// TwinCAT 3 PLC project Example_ExecutionToken
// ProgramVersion: 3.1.4024.0
// libraries:
//   Tc3_Module, * (Beckhoff Automation GmbH)
//   ZApplication, 1.6.0.6 (Zeugwerk GmbH)
//   ZAux, 1.6.0.6 (Zeugwerk GmbH)
//   ZCore, 1.6.0.6 (Zeugwerk GmbH)
//   ZEquipment, 1.6.0.6 (Zeugwerk GmbH)
//   ZPlatform, 1.6.0.6 (Zeugwerk GmbH)
// project tree:
//   ZApp/App/ ZApp.TcPOU
//   ZApp/App/_DataTypes/ ZAppStep.TcDUT
//   ZApp/App/_States/ ZAppSequenceBoot.TcPOU, ZAppSequenceBootFault.TcPOU, ZAppSequenceRunning.TcPOU
//   ZApp/App/_SubObjects/ ZAppSequence.TcPOU
//   ZApp/Com/_DataTypes/ ZCom.TcDUT, ZComUnit.TcDUT
//   ZApp/Data/_DataTypes/ ZData.TcDUT, ZDataMachine.TcDUT, ZDataConfig.TcDUT, ZDataCalibration.TcDUT, ZDataRecipe.TcDUT
//   ZApp/Unit/Picker/ IPicker.TcIO, PickerUnit.TcPOU, PickerUnitProgram.TcPOU
//   ZApp/Unit/Picker/_Com/ PickerCom.TcDUT, PickerComPublish.TcDUT, PickerComPublishEquipment.TcDUT, PickerComRef.TcDUT, PickerComRequest.TcDUT, PickerComSubscribe.TcDUT, PickerComSubscribeEquipment.TcDUT
//   ZApp/Unit/Picker/_DataTypes/ PickerState.TcDUT, PickerStep.TcDUT, PickerTokenUsage.TcDUT
//   ZApp/Unit/Picker/_Data/ PickerDataCalibration.TcDUT, PickerDataConfig.TcDUT, PickerDataMachine.TcDUT, PickerDataRef.TcDUT
//   ZApp/Unit/Picker/_Equipment/ PickerActuator.TcPOU, PickerAxis.TcPOU, PickerEquipment.TcPOU, PickerFieldbus.TcPOU, PickerIo.TcPOU, PickerLinkedUnit.TcPOU
//   ZApp/Unit/Picker/_States/ PickerSequenceAutomatic.TcPOU, PickerSequenceBoot.TcPOU, PickerSequenceFaultReaction.TcPOU, PickerSequenceGoHome.TcPOU, PickerSequenceStop.TcPOU
//   ZApp/Unit/Picker/_SubObjects/ PickerContainer.TcPOU, PickerSequence.TcPOU
//   ZApp/ ZGlobal.TcGVL, ZModuleProgram.TcPOU, ZModuleTask.TcTTO
// real-time tasks:
//   TASK ZModuleTask: cycle T#10ms, priority 20, ADS port 350

CONFIGURATION Example_ExecutionToken
    RESOURCE PLC ON TwinCAT3
        TASK ZModuleTask(INTERVAL := T#10ms, PRIORITY := 20);
        PROGRAM ZModuleProgram WITH ZModuleTask : ZModuleProgram;
    END_RESOURCE
END_CONFIGURATION

// ---- ZApp/App/_DataTypes/ZAppStep.TcDUT
{attribute 'qualified_only'}
{attribute 'to_string'}
TYPE ZAppStep :
(
  Undefined := 0
  
  ,BootBegin
  ,BootLoadDefaultData
  ,BootEnd
  ,BootFaultBegin
  ,BootFaultEnd 
  ,RunningBegin
  ,RunningEnd   
);
END_TYPE

// ---- ZApp/Com/_DataTypes/ZCom.TcDUT
TYPE ZCom :
STRUCT
  // module context
  App : ZApplication.ApplicationComPublish;
  Alarming : ZApplication.AlarmingCom;
  Messages : ZApplication.MessagingCom;
  
  // unit context
  Unit : ZComUnit;

END_STRUCT
END_TYPE

// ---- ZApp/Com/_DataTypes/ZComUnit.TcDUT
TYPE ZComUnit :
STRUCT
{region "Picker"}
{IF NOT (defined (Picker_disabled))}
  Picker : PickerCom;
  {attribute 'ZId' := 'c43c28b7-9e8c-48c6-a4f8-946be27888d3'}
{END_IF}
{endregion}
{attribute '__ZwPlcApplicationComUnitDeclaration__'} // Do not remove this attribute! It is used for code generation.
END_STRUCT
END_TYPE

// ---- ZApp/Data/_DataTypes/ZData.TcDUT
TYPE ZData :
STRUCT
  Config : ZDataConfig;
  Machine : ZDataMachine;
  Calibration : ZDataCalibration;
  Recipe : ZDataRecipe;
END_STRUCT
END_TYPE

// ---- ZApp/Data/_DataTypes/ZDataMachine.TcDUT
TYPE ZDataMachine :
STRUCT
{region "Picker"}
{IF NOT (defined (Picker_disabled))}
  Picker : PickerDataMachine;
  {attribute 'ZId' := 'c43c28b7-9e8c-48c6-a4f8-946be27888d3'}
{END_IF}
{endregion}
{attribute '__ZwPlcApplicationDataMachineDeclaration__'} // Do not remove this attribute! It is used for code generation.
END_STRUCT
END_TYPE

// ---- ZApp/Data/_DataTypes/ZDataConfig.TcDUT
TYPE ZDataConfig :
STRUCT
{region "Picker"}
{IF NOT (defined (Picker_disabled))}
  Picker : PickerDataConfig;
  {attribute 'ZId' := 'c43c28b7-9e8c-48c6-a4f8-946be27888d3'}
{END_IF}
{endregion}
{attribute '__ZwPlcApplicationDataConfigDeclaration__'} // Do not remove this attribute! It is used for code generation.
END_STRUCT
END_TYPE

// ---- ZApp/Data/_DataTypes/ZDataCalibration.TcDUT
TYPE ZDataCalibration :
STRUCT
{region "Picker"}
{IF NOT (defined (Picker_disabled))}
  Picker : PickerDataCalibration;
  {attribute 'ZId' := 'c43c28b7-9e8c-48c6-a4f8-946be27888d3'}
{END_IF}
{endregion}
{attribute '__ZwPlcApplicationDataCalibrationDeclaration__'} // Do not remove this attribute! It is used for code generation.
END_STRUCT
END_TYPE

// ---- ZApp/Data/_DataTypes/ZDataRecipe.TcDUT
TYPE ZDataRecipe :
STRUCT
  RecipeParam1 : LREAL;
  RecipeParam2 : LREAL;
  RecipeParam3 : LREAL;
END_STRUCT
END_TYPE

// ---- ZApp/Unit/Picker/_Com/PickerCom.TcDUT
/// This struct contains variables that
/// * are read from outside (e.g. HMI) to retrieve information about the unit's current state and (temporary) parameters (= `publish`) 
/// * are written from outside (e.g. HMI) to control the unit via ADS (= `subscribe`) 
TYPE PickerCom :
STRUCT
  Publish : PickerComPublish;
  Subscribe : PickerComSubscribe;
END_STRUCT
END_TYPE

// ---- ZApp/Unit/Picker/_Com/PickerComPublish.TcDUT
/// this is the container of informations that the unit wants to share with the world outside of the PLC
/// This struct should only be read from by external applications.
TYPE PickerComPublish :
STRUCT
  State : ZApplication.UnitStateMachineState; // state the unit is in
  Request : PickerComRequest; // booleans that indictate which action is currently possible to perform with this unit
  Equipment : PickerComPublishEquipment;  // structs for equipment objects which are used by the bridges
END_STRUCT
END_TYPE

// ---- ZApp/Unit/Picker/_Com/PickerComPublishEquipment.TcDUT
TYPE PickerComPublishEquipment :
STRUCT

{region "Vertical : Axis"}
  Vertical : ZApplication.AxisComPublish;
  {attribute 'ZId' := '1181714e-d83e-4cf6-aa91-287de19a3556'}
{endregion}

{attribute '__ZwPlcUnitComDeclaration__'} // Do not remove this attribute! It is used for code generation.

END_STRUCT
END_TYPE

// ---- ZApp/Unit/Picker/_Com/PickerComRef.TcDUT
/// container for all communication data types that are used by the unit
TYPE PickerComRef :
STRUCT
  Publish : REFERENCE TO PickerComPublish; 
  Subscribe : REFERENCE TO PickerComSubscribe; 
END_STRUCT
END_TYPE

// ---- ZApp/Unit/Picker/_Com/PickerComRequest.TcDUT
TYPE PickerComRequest :
STRUCT
  Start : BOOL;
  Stop : BOOL;
  GoHome : BOOL;
  Halt : BOOL;
END_STRUCT
END_TYPE

// ---- ZApp/Unit/Picker/_Com/PickerComSubscribe.TcDUT
TYPE PickerComSubscribe :
STRUCT
  Request : PickerComRequest; // contains booleans that are used to start a specific sequence.
  Equipment : PickerComSubscribeEquipment;  // structs for equipment objects which are used by the bridges
END_STRUCT
END_TYPE

// ---- ZApp/Unit/Picker/_Com/PickerComSubscribeEquipment.TcDUT
TYPE PickerComSubscribeEquipment :
STRUCT

{region "Vertical : Axis"}
  Vertical : ZApplication.AxisComSubscribe;
  {attribute 'ZId' := '1181714e-d83e-4cf6-aa91-287de19a3556'}
{endregion}

{attribute '__ZwPlcUnitComDeclaration__'} // Do not remove this attribute! It is used for code generation.

END_STRUCT
END_TYPE

// ---- ZApp/Unit/Picker/_DataTypes/PickerState.TcDUT
/// This enumeration contains all used defined sequences of a unit.
/// Per default a unit makes use of the states that are contained in (UnitStateDefault)[xref:ZApplication.UnitStateDefault]. However,
/// most of the time a unit need to perform some application depend sequences that can be performed by putting the unit into userdefined states.
/// For instance, a robotic unit could use the state (automatic)[xref:ZApplication.UnitStateDefault] to lift an object from point A to point B,
/// a userdefined state could be used to open and close the robotic-units gripper, respectively
{attribute 'qualified_only'}
TYPE PickerState :
(
	UserdefinedState1 := ZApplication.UnitStateMachineState.Last+1
);
END_TYPE

// ---- ZApp/Unit/Picker/_DataTypes/PickerStep.TcDUT
/// This enumeration contains all steps that are used by the various sequences of a unit.
/// Sequences use a subrange (***Begin to ***End) of this enumeration.
{attribute 'qualified_only'}
{attribute 'to_string'}
TYPE PickerStep :
(
  Undefined := 0
  
  ,BootBegin
  ,BootEnd 

  ,StopBegin
  ,StopEnd

  ,AutomaticBegin
  ,AutomaticEnd
  
  ,GoHomeBegin
  ,GoHomeMoveAxisTo60
  ,GoHomeMoveAxisBackTo0
  ,GoHomeEnd 
  
  ,FaultReactionBegin
  ,FaultReactionEnd
);
END_TYPE

// ---- ZApp/Unit/Picker/_DataTypes/PickerTokenUsage.TcDUT
{attribute 'qualified_only'}
TYPE PickerTokenUsage :
(
	StartToken
  ,ExecutionToken
  ,SequenceAsToken
);
END_TYPE

// ---- ZApp/Unit/Picker/_Data/PickerDataCalibration.TcDUT
/// calibration that is determined by calibration sequences of the unit (static offsets, shifts)
TYPE PickerDataCalibration :
STRUCT
END_STRUCT
END_TYPE

// ---- ZApp/Unit/Picker/_Data/PickerDataConfig.TcDUT
/// configuration data that is used during boot to configure the Units equipment
TYPE PickerDataConfig :
STRUCT
  Simulated : BOOL;
END_STRUCT
END_TYPE

// ---- ZApp/Unit/Picker/_Data/PickerDataMachine.TcDUT
/// machine data that is used through most sequences of the unit (motor speed, axes positions, ...)
TYPE PickerDataMachine :
STRUCT
  Slowspeed : LREAL;
  Highspeed : LREAL;
END_STRUCT
END_TYPE

// ---- ZApp/Unit/Picker/_Data/PickerDataRef.TcDUT
/// container for all data that are used by the unit
TYPE PickerDataRef :
STRUCT
  Config : REFERENCE TO PickerDataConfig; // data required for booting the unit (axes configuration, simulation, parameters that have to be written in PREOP, ...)
  Machine : REFERENCE TO PickerDataMachine; // speeds, positions, ...
  Calibration : REFERENCE TO PickerDataCalibration; // offsets, shifts of nominal to actual values
END_STRUCT
END_TYPE

// ---- ZApp/ZGlobal.TcGVL
{attribute 'qualified_only'}
VAR_GLOBAL
  Com : ZCom;
END_VAR
VAR_GLOBAL PERSISTENT
  Data : ZData;
END_VAR

// ---- ZApp/Unit/Picker/IPicker.TcIO
INTERFACE IPicker EXTENDS ZApplication.IUnit

END_INTERFACE

// ---- ZApp/ZModuleProgram.TcPOU
/// Zeugwerk Application
PROGRAM ZModuleProgram
VAR_INPUT
{region "ZModuleProgram : Utility"}
  App : ZApp(displayName:='Zeugwerk-Application Template', com:=ZGlobal.Com.App);
  Datetime : ZAux.DateTimeUM;
  {attribute 'ZId' := ''}
{endregion}
{region "ZModuleProgram : Logging"}
  Alarming : ZApplication.Alarming(App, datetime := Datetime, com := ZGlobal.Com.Alarming);
  LoggerHmi : ZApplication.Messaging(App, datetime := Datetime, com := ZGlobal.Com.Messages);
  LoggerFile : ZAux.LoggerFile7FF(App, datetime := Datetime, filePath:='C:\Zeugwerk\logs\messages.log', target:='');
  Logger : ZAux.Logging;
  {attribute 'ZId' := ''}
{endregion}  
{attribute '__ZwPlcApplicationModuleProgramDeclaration__'} // Do not remove this attribute! It is used for code generation.
{region "Picker"}
{undefine RunInSeparateProgram}
{IF NOT (defined (Picker_disabled)) AND NOT (defined (RunInSeparateProgram))}
  Picker : PickerUnit(displayName := 'Picker', // name of the unit (for logging)
					  parent := App, // caller of the Unit's cyclic method. If the Unit runs in its own context use 0
						configdata := ZGlobal.Data.Config.Picker,
						machinedata := ZGlobal.Data.Machine.Picker,
						calibrationdata := ZGlobal.Data.Calibration.Picker,
						com := ZGlobal.Com.Unit.Picker);
  {attribute 'section' := '__ZwPlcUnitProgramDeclaration__'}
  {attribute 'ZId' := 'c43c28b7-9e8c-48c6-a4f8-946be27888d3'}
{END_IF}
{endregion}
{attribute '__ZwPlcUnitProgramDeclaration__'} // Do not remove this attribute! It is used for code generation.
END_VAR

{region "ZModuleProgram : Utility"}
  Datetime.Cyclic();
  App.Cyclic();
  {attribute 'ZId' := ''}
{endregion}
{attribute '__ZwPlcApplicationModuleProgramImplementation__'} // Do not remove this attribute! It is used for code generation.

END_PROGRAM

// ---- ZApp/App/ZApp.TcPOU
FUNCTION_BLOCK ZApp EXTENDS ZApplication.Application
VAR
  _boot : ZAppSequenceBoot;
  _bootFault : ZAppSequenceBootFault;
  _running : ZAppSequenceRunning;
END_VAR

METHOD FB_init : BOOL
VAR_INPUT
  bInitRetains : BOOL; /// if TRUE, the retain variables are initialized (warm start / cold start)
  bInCopyCode : BOOL; /// if TRUE, the instance afterwards gets moved into the copy code (online change)
  displayName : ZCore.ZString;
  com : REFERENCE TO ZApplication.ApplicationComPublish;
END_VAR
SetBootSequence(_boot);
SetBootFaultSequence(_bootFault);
SetRunningSequence(_running);
END_METHOD

END_FUNCTION_BLOCK

// ---- ZApp/App/_States/ZAppSequenceBoot.TcPOU
FUNCTION_BLOCK ZAppSequenceBoot EXTENDS ZAppSequence IMPLEMENTS ZCore.ISequence
VAR
  _step : ZCore.Step(ZAppStep.BootBegin, ZAppStep.BootEnd);
END_VAR

IF OnStart(_step)
THEN
  // init custom sequence variables here ...
END_IF

REPEAT
  LogStep();

  CASE _step.Index OF
    (* -------------------------------------------------------------------------------------------------------------------------------- *)
    ZAppStep.BootBegin:
    (* -------------------------------------------------------------------------------------------------------------------------------- *)
    
      IF _step.OnEntry()
      THEN
        ZModuleProgram.LoggerFile.MinimumLevel := ZCore.LogLevel.Trace;
        ZModuleProgram.Logger.AddLogger(ZModuleProgram.LoggerFile);        
        {attribute '__ZwPlcAppZComModuleContext__'} // Do not remove this attribute! It is used for code generation.      
      END_IF
      
	  IF ZModuleProgram.Datetime.State <> ZCore.ObjectState.Booting
      THEN
        _step.SetNext(ZAppStep.BootLoadDefaultData);        
      END_IF
      
    (* -------------------------------------------------------------------------------------------------------------------------------- *)
    ZAppStep.BootLoadDefaultData:
    (* -------------------------------------------------------------------------------------------------------------------------------- *)

      {warning 'The application is loading the default config data on every restart!'}
      LoadDefaultConfigData();
      
      IF IsCommissioning()
      THEN
        LoadDefaultData();
      END_IF
      
      _step.SetNext(ZAppStep.BootEnd);
      
    (* -------------------------------------------------------------------------------------------------------------------------------- *)
    ZAppStep.BootEnd:
    (* -------------------------------------------------------------------------------------------------------------------------------- *)
      SetBusy(FALSE);
      
  ELSE
    Abort('sequence contains unhandled step');
  END_CASE
UNTIL _step.IsNotRepeatable() OR_ELSE NOT Busy END_REPEAT

METHOD  IsCommissioning : BOOL
IsCommissioning := TRUE;
END_METHOD

METHOD FINAL LoadDefaultConfigData

{region "Picker"}
  {IF NOT (defined (Picker_disabled))}
  ZGlobal.Data.Config.Picker.Simulated := TRUE;
  {region "UserInitCode"}
  // put your individual init code for this unit here
  {endregion}
  {END_IF}
  {attribute 'ZId' := 'c43c28b7-9e8c-48c6-a4f8-946be27888d3'}
{endregion}

{attribute '__ZwPlcUnitLoadDefaultConfigData__'} // Do not remove this attribute! It is used for code generation.
END_METHOD

METHOD FINAL LoadDefaultData

{attribute '__ZwPlcUnitLoadDefaultData__'} // Do not remove this attribute! It is used for code generation.
END_METHOD

END_FUNCTION_BLOCK

// ---- ZApp/App/_SubObjects/ZAppSequence.TcPOU
FUNCTION_BLOCK ABSTRACT ZAppSequence EXTENDS ZApplication.Sequence IMPLEMENTS ZCore.ISequence

METHOD StepDecoded : ZCore.ZString
VAR_INPUT
  stepIndex : INT;
END_VAR
VAR_INST
  _stepIndexDecoded : ZAppStep;
END_VAR
_stepIndexDecoded := stepIndex;
StepDecoded := TO_STRING(_stepIndexDecoded);
END_METHOD

END_FUNCTION_BLOCK

// ---- ZApp/App/_States/ZAppSequenceBootFault.TcPOU
FUNCTION_BLOCK ZAppSequenceBootFault EXTENDS ZAppSequence IMPLEMENTS ZCore.ISequence
VAR
  _step : ZCore.Step(ZAppStep.BootFaultBegin, ZAppStep.BootFaultEnd);
END_VAR

IF OnStart(_step)
THEN
  // init custom sequence variables here ...
END_IF

REPEAT
  LogStep();

  CASE _step.Index OF
    (* -------------------------------------------------------------------------------------------------------------------------------- *)
    ZAppStep.BootFaultBegin:
    (* -------------------------------------------------------------------------------------------------------------------------------- *)
      _step.SetNext(ZAppStep.BootFaultEnd);
      
    (* -------------------------------------------------------------------------------------------------------------------------------- *)
    ZAppStep.BootFaultEnd:
    (* -------------------------------------------------------------------------------------------------------------------------------- *)
      SetBusy(FALSE);
      
  ELSE
    Abort('sequence contains unhandled step');
  END_CASE
UNTIL _step.IsNotRepeatable() OR_ELSE NOT Busy END_REPEAT

END_FUNCTION_BLOCK

// ---- ZApp/App/_States/ZAppSequenceRunning.TcPOU
FUNCTION_BLOCK ZAppSequenceRunning EXTENDS ZAppSequence IMPLEMENTS ZCore.ISequence
VAR
  _step : ZCore.Step(ZAppStep.RunningBegin, ZAppStep.RunningEnd);
END_VAR

IF OnStart(_step)
THEN
  // init custom sequence variables here ...
END_IF

REPEAT
  LogStep();

  CASE _step.Index OF
    (* -------------------------------------------------------------------------------------------------------------------------------- *)
    ZAppStep.RunningBegin:
    (* -------------------------------------------------------------------------------------------------------------------------------- *)
      ; // implement me
      
    (* -------------------------------------------------------------------------------------------------------------------------------- *)
    ZAppStep.RunningEnd:
    (* -------------------------------------------------------------------------------------------------------------------------------- *)
      SetBusy(FALSE);
      
  ELSE
    Abort('sequence contains unhandled step');
  END_CASE
UNTIL _step.IsNotRepeatable() OR_ELSE NOT Busy END_REPEAT

END_FUNCTION_BLOCK

// ---- ZApp/Unit/Picker/PickerUnit.TcPOU
/// Declaration of a distinct unit of this application
FUNCTION_BLOCK PickerUnit EXTENDS ZApplication.Unit IMPLEMENTS IPicker
VAR
  _equipment : PickerEquipment(THIS^);
  _data : PickerDataRef;
  _com : PickerComRef;

  _boot : PickerSequenceBoot(THIS^);
  _automatic : PickerSequenceAutomatic(THIS^);
  _stop : PickerSequenceStop(THIS^);
  _gohome : PickerSequenceGoHome(THIS^);
  _faultReaction : PickerSequenceFaultReaction(THIS^);
  
  _statemachine : ZApplication.UnitStateMachine;

  _observeTimer : ZAux.Timer;
END_VAR

{attribute 'ZId' := '91d6f29c-305c-4899-88ef-1e5d578c2af4'}

IF _observeTimer.Done THEN
  _observeTimer.WaitAsync(0.1);
  
  // monitor _com for requested actions (e.g. start homing, start automatic mode, ...)
  ObserveRequest(_com.Subscribe.Request.Start, ZApplication.UnitStateMachineState.Automatic);
  ObserveRequest(_com.Subscribe.Request.Stop, ZApplication.UnitStateMachineState.Stop);
  ObserveRequest(_com.Subscribe.Request.GoHome, ZApplication.UnitStateMachineState.GoHome);
  ObserveRequest(_com.Subscribe.Request.Halt, ZApplication.UnitStateMachineState.Halt);
  
  // provide relevant information via ADS
  _com.Publish.Request.Stop := _stateMachine.IsTransitionAllowed(ZApplication.UnitStateMachineState.Stop);
  _com.Publish.Request.Start := _stateMachine.IsTransitionAllowed(ZApplication.UnitStateMachineState.Automatic);
  _com.Publish.Request.GoHome := _stateMachine.IsTransitionAllowed(ZApplication.UnitStateMachineState.GoHome);
  _com.Publish.Request.Halt := _stateMachine.IsTransitionAllowed(ZApplication.UnitStateMachineState.Halt);

  _com.Publish.State := _stateMachine.State();
END_IF

METHOD FB_init : BOOL
VAR_INPUT
  bInitRetains : BOOL; // if TRUE, the retain variables are initialized (warm start / cold start)
  bInCopyCode : BOOL;  // if TRUE, the instance afterwards gets moved into the copy code (online change)
  parent : ZCore.IManagedObject; // caller of the Unit's cyclic method. If the Unit runs in its own context use 0
  displayName : ZCore.ZString;  // name of this unit as it should show up in the logger
  configdata : REFERENCE TO PickerDataConfig;  // reference to the configuration data that is used during boot to configure the Units equipment
  machinedata : REFERENCE TO PickerDataMachine; // reference to the machine data that is used through most sequences of the unit (motor speed, axes positions, ...)
  calibrationdata : REFERENCE TO PickerDataCalibration;  // reference to calibration that is determined by calibration sequences of the unit (static offsets, shifts)
  com : REFERENCE TO PickerCom;  // reference to the communication interface that is used to control this Unit via ADS
END_VAR
_name := displayName;

// initialize local logger decorator
_loggerDecorator.FB_init(bInitRetains, bInCopyCode, _name, ZModuleProgram.Logger);
_alarmingDecorator.FB_init(bInitRetains, bInCopyCode, _name, ZModuleProgram.Alarming);

// setup data
_data.Config REF= configdata;
_data.Machine REF= machinedata;
_data.Calibration REF= calibrationdata;
_com.Publish REF= com.Publish;
_com.Subscribe REF= com.Subscribe;

// ------- sequence initialization, map sequences of this unit to the statemachine -------
{attribute '__ZwPlcUnitInitSequenceImplementation__'} // Do not remove this attribute! It is used for code generation.
_statemachine.SetSequence(ZApplication.UnitStateMachineState.Boot, _boot);
_statemachine.SetSequence(ZApplication.UnitStateMachineState.FaultReaction, _faultReaction);
_statemachine.SetSequence(ZApplication.UnitStateMachineState.Gohome, _gohome);
_statemachine.SetSequence(ZApplication.UnitStateMachineState.Stop, _stop);
_statemachine.SetSequence(ZApplication.UnitStateMachineState.Automatic, _automatic);

_statemachine.SetName(_name);
_statemachine.SetLogger(_logger);

// set initial state
_statemachine.SetState(ZApplication.UnitStateMachineState.Boot);
SetStateMachine(_statemachine);
END_METHOD

END_FUNCTION_BLOCK

// ---- ZApp/Unit/Picker/_Equipment/PickerEquipment.TcPOU
/// This function block is a container for equipment that is used by this unit.
/// Equipment is grouped by its kind (actuator, axes, io, ...).
/// It extends from [ManagedObjectContainer](xref:ZCore.ManagedObjectContainer) such that the parent
/// (= the unit itself) can be passed to equipment instances.
FUNCTION_BLOCK PickerEquipment EXTENDS PickerContainer
VAR_INPUT
  Io : PickerIo(_parent);
  Actuator : PickerActuator(_parent);
  Axis : PickerAxis(_parent);
  Fieldbus : PickerFieldbus(_parent);
  Unit : PickerLinkedUnit(_parent);
END_VAR

END_FUNCTION_BLOCK

// ---- ZApp/Unit/Picker/_SubObjects/PickerContainer.TcPOU
FUNCTION_BLOCK PickerContainer EXTENDS ZCore.ObjectContainer
VAR_INPUT
END_VAR
VAR_OUTPUT
END_VAR
VAR
  {attribute 'hide'}
  _parent : REFERENCE TO PickerUnit;
END_VAR

{attribute 'hide' }
METHOD FB_init : BOOL
VAR_INPUT
	bInitRetains : BOOL; // if TRUE, the retain variables are initialized (warm start / cold start)
	bInCopyCode : BOOL;  // if TRUE, the instance afterwards gets moved into the copy code (online change)
  unit : REFERENCE TO PickerUnit;
END_VAR
_parent REF= unit;
END_METHOD

END_FUNCTION_BLOCK

// ---- ZApp/Unit/Picker/_Equipment/PickerIo.TcPOU
/// This function block is a container for all I/Os that are used by this unit.
/// The parent of all objects can be directly transfered in their constructor (this is only relevant for equipment objects
/// that have to be managed (e.g. [DebouncedInput](xref:ZEquipment.DebouncedInput), [Light](xref:ZEquipment.Light), ...).
FUNCTION_BLOCK PickerIo EXTENDS PickerContainer
VAR
  {attribute 'hide'}
  _iobridge : ZApplication.IoBridge(_parent);
END_VAR
VAR_INPUT

{attribute '__ZwPlcUnitEquipmentDeclaration__'} // Do not remove this attribute! It is used for code generation.
END_VAR

IF _isInitialized
THEN
  RETURN;
END_IF

  _iobridge.SetLogger(_parent._logger);

{attribute '__ZwPlcUnitEquipmentImplementation__'} // Do not remove this attribute! It is used for code generation.

_isInitialized := TRUE;

END_FUNCTION_BLOCK

// ---- ZApp/Unit/Picker/_Equipment/PickerActuator.TcPOU
/// This function block is a container for all actuator objects that are used by this unit.
/// The parent of all objects can be directly transfered in their constructor (this is only relevant for equipment objects
/// that have to be managed (e.g. [DebouncedInput](xref:ZEquipment.DebouncedInput), [Light](xref:ZEquipment.Light), ...).
FUNCTION_BLOCK PickerActuator EXTENDS PickerContainer
VAR
  {attribute 'hide'}
  _actuatorbridge : ZApplication.ActuatorBridge(_parent);
  {attribute 'hide'}
  _iobridge : ZApplication.IoBridge(_parent);
END_VAR
VAR_INPUT

{attribute '__ZwPlcUnitEquipmentDeclaration__'} // Do not remove this attribute! It is used for code generation.
END_VAR

IF _isInitialized
THEN
  RETURN;
END_IF

  _actuatorbridge.SetLogger(_parent._logger);

{attribute '__ZwPlcUnitEquipmentImplementation__'} // Do not remove this attribute! It is used for code generation.

_isInitialized := TRUE;

END_FUNCTION_BLOCK

// ---- ZApp/Unit/Picker/_Equipment/PickerAxis.TcPOU
/// This function block is a container for all axis objects that are used by this unit.
/// The parent of all objects can be directly transfered in their constructor (this is only relevant for equipment objects
/// that have to be managed (e.g. [DebouncedInput](xref:ZEquipment.DebouncedInput), [Light](xref:ZEquipment.Light), ...).
FUNCTION_BLOCK PickerAxis EXTENDS PickerContainer
VAR
  {attribute 'hide'}
  _axisbridge : ZApplication.AxisBridge(_parent);
END_VAR
VAR_INPUT

{region "Vertical : AxisPlcOpenMc"}
  Vertical : ZEquipment.AxisPlcOpenMc(_parent);
  {attribute 'ZId' := '1181714e-d83e-4cf6-aa91-287de19a3556'}
{endregion}

{attribute '__ZwPlcUnitEquipmentDeclaration__'} // Do not remove this attribute! It is used for code generation.
END_VAR

IF _isInitialized
THEN
  RETURN;
END_IF

  _axisbridge.SetLogger(_parent._logger);

{region "Vertical : AxisPlcOpenMc"}
  Vertical.SetLogger(_parent._logger);
  Vertical.SetName(name:='Vertical');
  Vertical.SetSimulation(_parent._data.Config.Simulated);
  _axisbridge.AddAxisPlcOpenMc(axis:=Vertical, publish:=_parent._com.Publish.Equipment.Vertical, subscribe:=_parent._com.Subscribe.Equipment.Vertical);

  {region "UserInitCode"}
  // put your individual init code for this Axis here
  {endregion}

  {attribute 'ZId' := '1181714e-d83e-4cf6-aa91-287de19a3556'}
{endregion}

{attribute '__ZwPlcUnitEquipmentImplementation__'} // Do not remove this attribute! It is used for code generation.

_isInitialized := TRUE;

END_FUNCTION_BLOCK

// ---- ZApp/Unit/Picker/_Equipment/PickerFieldbus.TcPOU
/// This function block is a container for all axis objects that are used by this unit.
/// The parent of all objects can be directly transfered in their constructor (this is only relevant for equipment objects
/// that have to be managed (e.g. [DebouncedInput](xref:ZEquipment.DebouncedInput), [Light](xref:ZEquipment.Light), ...).
FUNCTION_BLOCK PickerFieldbus EXTENDS PickerContainer
VAR
END_VAR
VAR_INPUT

{attribute '__ZwPlcUnitEquipmentDeclaration__'} // Do not remove this attribute! It is used for code generation.
END_VAR

IF _isInitialized
THEN
  RETURN;
END_IF

{attribute '__ZwPlcUnitEquipmentImplementation__'} // Do not remove this attribute! It is used for code generation.

_isInitialized := TRUE;

END_FUNCTION_BLOCK

// ---- ZApp/Unit/Picker/_Equipment/PickerLinkedUnit.TcPOU
/// This function block is a container for all linked units that are used by this unit.
/// Linked units can be addressed through their individual interface.
FUNCTION_BLOCK PickerLinkedUnit EXTENDS PickerContainer
VAR_INPUT

{attribute '__ZwPlcUnitEquipmentDeclaration__'} // Do not remove this attribute! It is used for code generation.
END_VAR

IF _isInitialized
THEN
  RETURN;
END_IF

{attribute '__ZwPlcUnitEquipmentImplementation__'} // Do not remove this attribute! It is used for code generation.

_isInitialized := TRUE;

END_FUNCTION_BLOCK

// ---- ZApp/Unit/Picker/_States/PickerSequenceBoot.TcPOU
FUNCTION_BLOCK PickerSequenceBoot EXTENDS PickerSequence IMPLEMENTS ZCore.ISequence
VAR
  _step : ZCore.Step(PickerStep.BootBegin, PickerStep.BootEnd);
END_VAR

IF OnStart(_step) THEN
  ; // init custom sequence variables here ...
END_IF

REPEAT
  LogStep();

  CASE _step.Index OF
    (* -------------------------------------------------------------------------------------------------------------------------------- *)
    PickerStep.BootBegin:
    (* -------------------------------------------------------------------------------------------------------------------------------- *)
      IF _step.OnEntry()
      THEN
        // initialize equipment
        _io();
        _actuator();
        _fieldbus();
        _axis();
        _unit();
      END_IF
      
      _parent._objectManager.Cyclic();      
      Assert(_parent._objectManager);
      IF _parent._objectManager.Booted
      THEN
        _step.SetNext(PickerStep.BootEnd);
      END_IF

    (* -------------------------------------------------------------------------------------------------------------------------------- *)
    PickerStep.BootEnd:
    (* -------------------------------------------------------------------------------------------------------------------------------- *)
      SetBusy(FALSE);
      
  ELSE
    Abort('sequence contains unhandled step');
  END_CASE
UNTIL _step.IsNotRepeatable() OR_ELSE NOT Busy END_REPEAT

END_FUNCTION_BLOCK

// ---- ZApp/Unit/Picker/_SubObjects/PickerSequence.TcPOU
FUNCTION_BLOCK PickerSequence EXTENDS ZApplication.Sequence
VAR
  {attribute 'hide'}
  _parent : REFERENCE TO PickerUnit;
  _io : REFERENCE TO PickerIo;
  _actuator : REFERENCE TO PickerActuator;
  _fieldbus : REFERENCE TO PickerFieldbus;
  _axis : REFERENCE TO PickerAxis;
  _data : REFERENCE TO PickerDataRef;
  _unit : REFERENCE TO PickerLinkedUnit;  
END_VAR

METHOD FB_init : BOOL
VAR_INPUT
  bInitRetains : BOOL; // if TRUE, the retain variables are initialized (warm start / cold start)
  bInCopyCode : BOOL;  // if TRUE, the instance afterwards gets moved into the copy code (online change)
  unit : REFERENCE TO PickerUnit;
END_VAR
_parent REF= unit;
_alarming := unit._alarming;
_io REF= unit._equipment.Io;
_actuator REF= unit._equipment.Actuator;
_fieldbus REF= unit._equipment.Fieldbus;
_axis REF= unit._equipment.Axis;
_unit REF= unit._equipment.Unit;
_data REF= unit._data;
_loggerDiagnostics.SetLogger(unit._logger);
END_METHOD

METHOD StepDecoded : ZCore.ZString
VAR_INPUT
  stepIndex : INT;
END_VAR
VAR_INST
  _stepIndexDecoded : PickerStep;
END_VAR
_stepIndexDecoded := stepIndex;
stepDecoded := TO_STRING(_stepIndexDecoded);
END_METHOD

END_FUNCTION_BLOCK

// ---- ZApp/Unit/Picker/_States/PickerSequenceAutomatic.TcPOU
FUNCTION_BLOCK PickerSequenceAutomatic EXTENDS PickerSequence IMPLEMENTS ZCore.ISequence
VAR
  _step : ZCore.Step(PickerStep.AutomaticBegin, PickerStep.AutomaticEnd);
END_VAR

IF NOT Busy THEN
  RETURN;
END_IF

IF OnStart(_step) THEN
  ; // init custom sequence variables here ...
END_IF

IF OnStop() THEN
  RETURN; // external stop was triggered
END_IF

IF OnHalt() THEN
  ; // Halting := TRUE; // Uncomment to acknowledge that the sequence is halting
END_IF

REPEAT
  LogStep();

  CASE _step.Index OF
    (* -------------------------------------------------------------------------------------------------------------------------------- *)
    PickerStep.AutomaticBegin:
    (* -------------------------------------------------------------------------------------------------------------------------------- *)
      IF _step.OnEntry()
      THEN
        ;
      END_IF

      // Await(obj1:=, nextStep:=PickerStep.AutomaticEnd);
      _step.SetNext(PickerStep.AutomaticEnd);
    
    (* -------------------------------------------------------------------------------------------------------------------------------- *)
    PickerStep.AutomaticEnd:
    (* -------------------------------------------------------------------------------------------------------------------------------- *)
      SetBusy(FALSE);
  
  ELSE
    Abort('sequence contains unhandled step');
  END_CASE
UNTIL _step.IsNotRepeatable() OR_ELSE NOT Busy END_REPEAT

END_FUNCTION_BLOCK

// ---- ZApp/Unit/Picker/_States/PickerSequenceStop.TcPOU
FUNCTION_BLOCK PickerSequenceStop EXTENDS PickerSequence IMPLEMENTS ZCore.ISequence
VAR
  _step : ZCore.Step(PickerStep.StopBegin, PickerStep.StopEnd);
  _timerSim : ZAux.Timer;
END_VAR

IF OnStart(_step) THEN
  ; // init custom sequence variables here ...
END_IF

REPEAT
  LogStep();

  CASE _step.Index OF
    (* -------------------------------------------------------------------------------------------------------------------------------- *)
    PickerStep.StopBegin:
    (* -------------------------------------------------------------------------------------------------------------------------------- *)
      IF _step.OnEntry()
      THEN
        _timerSim.WaitAsync(5);
			END_IF
      
      Await(_timerSim, nextStep:=PickerStep.StopEnd);
      // _step.SetNext(index:=PickerStep.StopEnd);

    (* -------------------------------------------------------------------------------------------------------------------------------- *)
    PickerStep.StopEnd:
    (* -------------------------------------------------------------------------------------------------------------------------------- *)    
      SetBusy(FALSE);
  
  ELSE
    Abort('sequence contains unhandled step');
  END_CASE
UNTIL _step.IsNotRepeatable() OR_ELSE NOT Busy END_REPEAT

END_FUNCTION_BLOCK

// ---- ZApp/Unit/Picker/_States/PickerSequenceGoHome.TcPOU
/// "Async" methods accept an IStartToken parameter to indicate whether 
/// the method was executed successfully. Additional to the StartToken, 
/// an ZCore.ExcecutionToken is now available to not only check if the 
/// method call was successful, but also to monitor the whole execution 
/// of the task. The ExecutionToken gets informed (aborted), if the 
/// originally started task changed unexpected.
FUNCTION_BLOCK PickerSequenceGoHome EXTENDS PickerSequence IMPLEMENTS ZCore.ISequence
VAR
  _step : ZCore.Step(PickerStep.GohomeBegin, PickerStep.GohomeEnd);
  _timer : ZAux.Timer;
  
  _startToken : ZCore.StartToken;
  _executionToken : ZCore.ExecutionToken;
  
  // Change this value to see what happens with differnt objects used as the startToken parameter
  _tokenUsage : PickerTokenUsage := PickerTokenUsage.StartToken;
  
  _usedToken : ZCore.IStartToken;
END_VAR

IF NOT Busy THEN
  RETURN;
END_IF

IF OnStart(_step) THEN
  ; // init custom sequence variables here ...
END_IF

IF OnStop() THEN
  RETURN; // external stop was triggered
END_IF

IF OnHalt() THEN
  ; // Halting := TRUE; // Uncomment to acknowledge that the sequence is halting
END_IF

REPEAT
  LogStep();

  CASE _step.Index OF
    (* -------------------------------------------------------------------------------------------------------------------------------- *)
    PickerStep.GoHomeBegin:
    (* -------------------------------------------------------------------------------------------------------------------------------- *)
      IF _step.OnEntry()
      THEN      
        // move to 0 initially
        _axis.Vertical.MoveAbsoluteAsync(THIS^, 0, 100);        
			END_IF
      
      Await(_axis.Vertical, nextStep:=PickerStep.GoHomeMoveAxisTo60);

    (* -------------------------------------------------------------------------------------------------------------------------------- *)
    PickerStep.GoHomeMoveAxisTo60:
    (* -------------------------------------------------------------------------------------------------------------------------------- *)
      IF _step.OnEntry()
      THEN        
        // ~~~~~~~~~~~~~~~~~~~~~~~~~~~~~~~~~~~~~~~~~~~~~~~~~~~~~~~~~~~~~
        // Choose the token to be used as the startToken for the Async call
        // ~~~~~~~~~~~~~~~~~~~~~~~~~~~~~~~~~~~~~~~~~~~~~~~~~~~~~~~~~~~~~   
        _startToken.Recover();
        _executionToken.Recover();            
        CASE _tokenUsage OF
          PickerTokenUsage.StartToken:      _usedToken := _startToken;
          PickerTokenUsage.ExecutionToken:  _usedToken := _executionToken;
          PickerTokenUsage.SequenceAsToken: _usedToken := THIS^;
				END_CASE

        _timer.WaitAsync(2);
        
        // start moving to 30
        _axis.Vertical.MoveAbsoluteAsync(_usedToken, 30, 10);
      END_IF
      
      IF _timer.OnDone() THEN
        // ~~~~~~~~~~~~~~~~~~~~~~~~~~~~~~~~~~~~~~~~~~~~~~~~~~~~~~~~~~~~~
        // Change the target position after 2 seconds --> no problem, 
        // because by using the same token you make a deliberate change
        // of the originally task.
        // ~~~~~~~~~~~~~~~~~~~~~~~~~~~~~~~~~~~~~~~~~~~~~~~~~~~~~~~~~~~~~   
        _axis.Vertical.MoveAbsoluteAsync(_usedToken, 60, 10);
			END_IF
      
      Await(obj1:=_axis.Vertical, nextStep:=PickerStep.GoHomeMoveAxisBackTo0);

    (* -------------------------------------------------------------------------------------------------------------------------------- *)
    PickerStep.GoHomeMoveAxisBackTo0:
    (* -------------------------------------------------------------------------------------------------------------------------------- *)
      IF _step.OnEntry()
      THEN        
        _timer.WaitAsync(2);
        
        // start moving to 0
        _axis.Vertical.MoveAbsoluteAsync(_usedToken, 0, 10);
      END_IF
      
      IF _timer.OnDone() THEN
        // stop the axis after 2 seconds without token - this is an unexpected change of the originally started MoveAbsoluteAsync task.
        _axis.Vertical.StopAsync(0);
        
        // ~~~~~~~~~~~~~~~~~~~~~~~~~~~~~~~~~~~~~~~~~~~~~~~~~~~~~~~~~~~~~
        // What happens depends on the token which was used to start the Movement!
        //
        // Using the _startToken (ZCore.StartToken):
        //   The change is not recognized by the sequence, as the StartToken is only 
        //   used by Async methods to indicate whether the method call was successful.
        //   After Stop is finished, the sequence continues with the next step as
        //   the axis changes to Idle.
        //
        // Using the _executionToken (ZCore.ExecutionToken):
        //   The change is recognized by the _executionToken, as the ExecutionToken is 
        //   additionally to the StartToken used to monitor unexpected changes of the 
        //   originally started task.
        //
        // Using the sequence (THIS^):
        //   A sequence is a ZCore.ExecutionToken.
        //   The change is automatically recognized by the sequence, as it is aborted
        //   when the unexpected change occurs. You have nothing to do, the sequence
        //   is in Error state an will be ended as if you would call Abort().  
        // ~~~~~~~~~~~~~~~~~~~~~~~~~~~~~~~~~~~~~~~~~~~~~~~~~~~~~~~~~~~~~               
        
			END_IF
      
      // If an ExecutionToken is used, you can observe it to recognize an unexpected change of the originally started task
      IF NOT Assert(_executionToken) THEN
        _logger.Error('The ExecutionToken used to monitor the movement was informed of an unexpected change');
      ELSIF Error THEN
        _logger.Error('The Sequence used to monitor the movement was informed of an unexpected change');
			END_IF
      
      Await(obj1:=_axis.Vertical, nextStep:=PickerStep.GoHomeEnd);

    (* -------------------------------------------------------------------------------------------------------------------------------- *)
    PickerStep.GoHomeEnd:
    (* -------------------------------------------------------------------------------------------------------------------------------- *)
      SetBusy(FALSE);
  
  ELSE
    Abort('sequence contains unhandled step');
  END_CASE
UNTIL _step.IsNotRepeatable() OR_ELSE NOT Busy END_REPEAT

END_FUNCTION_BLOCK

// ---- ZApp/Unit/Picker/_States/PickerSequenceFaultReaction.TcPOU
FUNCTION_BLOCK PickerSequenceFaultReaction EXTENDS PickerSequence IMPLEMENTS ZCore.ISequence
VAR
  _step : ZCore.Step(PickerStep.FaultReactionBegin, PickerStep.FaultReactionEnd);
  _timerSim : ZAux.Timer;
END_VAR

IF OnStart(_step) THEN
  ; // init custom sequence variables here ...
END_IF

REPEAT
  LogStep();

  CASE _step.Index OF
    (* -------------------------------------------------------------------------------------------------------------------------------- *)
    PickerStep.FaultReactionBegin:
    (* -------------------------------------------------------------------------------------------------------------------------------- *)
      IF _step.OnEntry()
      THEN
        _timerSim.WaitAsync(5);
			END_IF
      
      Await(_timerSim, nextStep:=PickerStep.FaultReactionEnd);
      // _step.SetNext(index:=PickerStep.FaultReactionEnd);

    (* -------------------------------------------------------------------------------------------------------------------------------- *)
    PickerStep.FaultReactionEnd:
    (* -------------------------------------------------------------------------------------------------------------------------------- *)    
      SetBusy(FALSE);
  
  ELSE
    Abort('sequence contains unhandled step');
  END_CASE
UNTIL _step.IsNotRepeatable() OR_ELSE NOT Busy END_REPEAT

END_FUNCTION_BLOCK

// ---- ZApp/Unit/Picker/PickerUnitProgram.TcPOU
/// each unit can run in its own PROGRAM and Task, respectively. However, this is optional and one may also
/// instantiate the unit in the ModuleProgram.
/// In order to keep initialization to a minimum, all ModuleContext objects that are required by the Unit are
/// given as FB_init parameter. These objects are
/// * data structs
/// * communication structs
/// * busmaster(s)
/// A unit should always be a root object (no parent) if it is running in its own context. If it runs in the same
/// task as the Module the parent may be set to the Module's Application.
PROGRAM PickerUnitProgram
VAR
{region "Picker"}
{undefine RunInSeparateProgram}
{IF NOT (defined (Picker_disabled)) AND (defined (RunInSeparateProgram))}
  Picker : PickerUnit(displayName := 'Picker', // name of the unit (for logging)
					  parent := 0, // caller of the Unit's cyclic method. If the Unit runs in its own context use 0
						configdata := ZGlobal.Data.Config.Picker,
						machinedata := ZGlobal.Data.Machine.Picker,
						calibrationdata := ZGlobal.Data.Calibration.Picker,
						com := ZGlobal.Com.Unit.Picker);
  {attribute 'section' := '__ZwPlcUnitProgramDeclaration__'}
  {attribute 'ZId' := 'c43c28b7-9e8c-48c6-a4f8-946be27888d3'}
{END_IF}
{endregion}
{attribute '__ZwPlcUnitProgramDeclaration__'} // Do not remove this attribute! It is used for code generation.
END_VAR

// run the unit - the cylics of all children will be called as well

{region "Picker"}
{undefine RunInSeparateProgram}
{IF NOT (defined (Picker_disabled)) AND (defined (RunInSeparateProgram))}
  Picker.Cyclic();
  {attribute 'section' := '__ZwPlcUnitProgramImplementation__'}
  {attribute 'ZId' := 'c43c28b7-9e8c-48c6-a4f8-946be27888d3'}
{END_IF}
{endregion}
{attribute '__ZwPlcUnitProgramImplementation__'} // Do not remove this attribute! It is used for code generation.

END_PROGRAM
